PROGRAM MAIN
VAR
	fbEcCoeSdoRead : FB_EcCoESdoRead;
	torque : REAL;
END_VAR

fbEcCoeSdoRead(
	sNetId:= '10.200.128.47.2.1', 
	nSlaveAddr:= 1002, 
	nSubIndex:=  17, 
	nIndex:= 16#32C0, 
	pDstBuf:= ADR(torque), 
	cbBufLen:= SIZEOF(torque), 
	bExecute:= , 
	);

END_PROGRAM

(* stored: Version 1.1.0.1
   POU MAIN: Id {b5d9e6a3-c16f-4431-a0e6-6d655d0029d2}, SpecialFunc None *)
